// TIA Portal V21 export
TYPE "LBC_typeAnalogInputInterface"
TITLE = LBC_typeAnalogInputInterface
// Module interface for external systems
   STRUCT
      commands : "LBC_typeInterfaceCommands";
      monitoring { ExternalWritable := 'False'} : "LBC_typeAnalogProcessValues";
      configuration : "LBC_typeAnalogInputConfiguration";
   END_STRUCT;
END_TYPE
